// TIA Portal project "snag7_test" (V18)

(* hardware
DEVICE "S7-1200-Station_1"  S7-1200 Station
   slot 0: "Baugruppenträger_0"  S7-1200 Rack  Rack  V1.0
   slot 1: "PLC_1"  CPU 1212C DC/DC/DC  6ES7 212-1AE40-0XB0  V4.6
*)

// ===== PLC "PLC_1"  CPU 1212C DC/DC/DC =====

DATA_BLOCK "test_db"   // DB1
{ S7_Optimized_Access := 'FALSE' }
VERSION : 0.1
   VAR
      vx_scaled : Real := 4.0;
      vy_scaled : Real := 5.0;
      vz_scaled : Real := 6.0;
      bool_1 : Bool;
      bool_2 : Bool := true;
      bool_3 : Bool := true;
      bool_4 : Bool;
      int_1 : Int := 32;
      int_2 : Int := 211;
   END_VAR
BEGIN
END_DATA_BLOCK

ORGANIZATION_BLOCK "Main"   // OB1, LAD, ProgramCycle
TITLE = "Main Program Sweep (Cycle)"
{ S7_Optimized_Access := 'TRUE' }
VERSION : 0.1
   VAR_INPUT
      Initial_Call : Bool;   // Initial call of this OB
      Remanence : Bool;   // =True, if remanent data are available
   END_VAR
BEGIN
END_ORGANIZATION_BLOCK